//These are variables every PLC project should have
VAR_GLOBAL

    stSys	:	ST_System; //Included for you
    fTimeStamp: LREAL;
END_VAR

(* stored: Version 1.1.0.1, ProductVersion 3.1.4022.12
   GVL DefaultGlobals: Id {2d2569a9-cdb9-4b2c-9048-e9448cd0d09e} *)
